Yaskawa INFORM job: R2_W39(90,0)AWOK.JBI

/JOB
//NAME R2_W39(90,0)AWOK
///FOLDERNAME AWOK
//POS
///NPOS 36,36,0,2,0,0
///TOOL 0
///POSTYPE PULSE
///PULSE
C00000=48919,5665,-78085,33957,84829,-60043
C00001=76192,72700,-3611,7580,89499,-58244
C00002=80540,137269,86328,-8121,96898,-60749
C00003=80542,135446,87907,-8083,95008,-60625
C00004=80542,134862,88738,-8070,94204,-60573
C00005=80542,134608,89189,-8064,93800,-60546
C00006=80542,134862,88738,-8070,94204,-60573
C00007=80678,141721,101118,-24359,107834,-67969
C00008=80550,135038,103284,-37220,113287,-73336
C00009=80378,131351,98751,-37526,113933,-73663
C00010=80550,135038,103284,-37220,113287,-73336
C00011=80547,133645,97127,919,61293,-41782
C00012=80548,133707,97515,920,61086,-41784
C00013=80548,134275,100610,935,59473,-41797
C00014=80549,134286,100620,934,59472,-41797
C00015=80548,134275,100610,935,59473,-41797
C00016=80547,133599,96697,917,61534,-41780
C00017=80549,133856,98384,924,60628,-41787
C00018=80549,133649,96859,917,61460,-41780
C00019=80548,133561,93639,902,63396,-41765
C00020=80524,99286,38399,14384,108927,-2349
C00021=80525,97179,39299,14231,107340,-2544
C00022=80951,95250,38355,13420,106584,-2631
C00023=80348,95814,37890,14264,107528,-2580
C00024=80254,94172,37553,14217,106925,-2684
C00025=80319,95343,39475,19204,110654,-13414
C00026=80535,96727,39662,19290,111179,-13264
C00027=80533,98698,38722,19533,112685,-13001
C00028=95804,88670,27983,-9101,104845,39456
C00029=95125,121930,72974,-13232,104168,56767
C00030=97567,93704,40848,-13739,109674,56976
C00031=97503,98351,37938,-14194,113675,56454
C00032=98256,60414,-24459,-19511,102185,56251
C00033=69963,28472,-55800,11354,92225,-11117
C00034=61683,17043,-76984,-12013,99317,-2721
C00035=8337,141,-97195,-54,99052,-6651
BC00000=111331,183388,1075175
BC00001=111331,183388,1075175
BC00002=111331,183388,1075175
BC00003=109903,183515,1075175
BC00004=109332,183566,1075175
BC00005=109318,182621,1075175
BC00006=109332,183566,1075175
BC00007=103421,136681,1075175
BC00008=99487,105483,1075175
BC00009=99485,107426,1074375
BC00010=99487,105483,1075175
BC00011=103771,236662,1075175
BC00012=103795,240102,1075175
BC00013=103795,240102,1075175
BC00014=102267,240107,1075175
BC00015=103795,240102,1075175
BC00016=103770,236662,1075175
BC00017=98594,239003,1075175
BC00018=98802,241035,1075175
BC00019=99321,246116,1075175
BC00020=156339,189130,1075175
BC00021=156280,185003,1075175
BC00022=156270,184325,1075174
BC00023=156256,183353,1075175
BC00024=156256,183353,1075175
BC00025=132811,179422,1075175
BC00026=133619,181005,1075175
BC00027=135738,184984,1075175
BC00028=156256,183353,1075175
BC00029=156256,183353,1075171
BC00030=156256,183353,1075171
BC00031=156256,183353,1075171
BC00032=156256,183353,1075171
BC00033=130207,183373,1075173
BC00034=130207,183373,1075173
BC00035=130207,258017,1075173
///POSTYPE BASE
///RECTAN
///RCONF 0,0,0,0,0,0,0,0,0,0,0,0,0,0,0,0,0,0,0,0,0,0,0,0
P00006=0.222,-3.123,-1.508,0.0000,0.0000,0.0000
P00022=0.222,-3.123,-1.508,0.0000,0.0000,0.0000
//INST
///DATE 2023/11/16 10:46
///ATTR SC,RW
///GROUP1 RB1,BS1
NOP
'r2_W39(90,0)
'Path S818
MOVJ C00000 BC00000 VJ=20.00
MOVJ C00001 BC00001 VJ=20.00
SFTOF
MOVJ C00002 BC00002 VJ=20.00
MOVL C00003 BC00003 V=100.0
MOVL C00004 BC00004 V=60.0
REFP 3 C00005 BC00005
CALL JOB:SEARCH-R1
SET P022 P006
SFTON P022
MOVL C00006 BC00006 V=60.0
MOVL C00007 BC00007 V=100.0
MOVL C00008 BC00008 V=60.0
REFP 3 C00009 BC00009
CALL JOB:SEARCH-R1
SET P022 P006
SFTON P022
MOVL C00010 BC00010 V=60.0
MOVL C00011 BC00011 V=100.0
MOVL C00012 BC00012 V=100.0
MOVL C00013 BC00013 V=60.0
REFP 3 C00014 BC00014
CALL JOB:SEARCH-R1
SET P022 P006
SFTON P022
MOVL C00015 BC00015 V=60.0
MOVL C00016 BC00016 V=100.0
MOVL C00017 BC00017 V=100.0
MOVL C00018 BC00018 V=100.0
MOVL C00019 BC00019 V=100.0
'Path W73
SFTOF
SFTON P022
MOVJ C00020 BC00020 VJ=20.00
MOVL C00021 BC00021 V=100.0
MOVL C00022 BC00022 V=100.0 PL=0
REFP 1 C00023 BC00023
REFP 2 C00024 BC00024
MACRO1 MJ#(0) ARGF10
ARCON
MOVL C00025 BC00025 V=15.0
ARCOF
MOVL C00026 BC00026 V=100.0
MOVL C00027 BC00027 V=100.0
SFTOF
'COMMENT
SFTON P022
MOVL C00028 BC00028 V=100.0
MOVL C00029 BC00029 V=100.0 PL=0
MACRO1 MJ#(0) ARGF10
ARCON
MOVL C00030 BC00030 V=15.0
ARCOF
SFTOF
MOVL C00031 BC00031 V=100.0
MOVJ C00032 BC00032 VJ=20.00
MOVJ C00033 BC00033 VJ=20.00
MOVJ C00034 BC00034 VJ=20.00
MOVJ C00035 BC00035 VJ=20.00
SFTOF
END
